FUNCTION_BLOCK FB_PointCorr
VAR PERSISTENT
  _fX_Pos, _fX_Ref : LREAL;   // x position (correction / reference)
  _fY_Pos, _fY_Ref : LREAL;   // y position (correction / reference)
END_VAR
VAR
  bCmd_X_minus : BOOL;    // command x minus
  bCmd_X_plus  : BOOL;    // command x plus
  bCmd_Y_minus : BOOL;    // command y minus
  bCmd_Y_plus  : BOOL;    // command y plus
  bAny         : BOOL;    // any pressed
  tSlow, tFast : TON;
  rTrig        : R_TRIG;
  nIncr        : LREAL;
  nBtnColor    : UDINT;
  // settings (init)
  _aName       : STRING(3);   // name of element
  _aUnit       : STRING(10);  // element intended [unit]
  _fX_Min, _fX_Max : LREAL;   // limit x
  _fY_Min, _fY_Max : LREAL;   // limit y
  _fIncrStep    : LREAL;      // incr. step slow (stay on button), fast *10
  _bButnInvertX, _bButnInvertY : BOOL;  // change buttons
  _bValInvertX, _bValInvertY   : BOOL;  // value *-1
END_VAR
VAR CONSTANT
  RED          : UDINT := 16#FFFF0000;
  GREEN        : UDINT := 16#FF00FF00;
END_VAR

bAny := bCmd_X_minus OR bCmd_X_plus OR bCmd_Y_minus OR bCmd_Y_plus;
rTrig(CLK:=bAny);
tSlow(IN:=bAny AND NOT tSlow.Q, PT:=T#500MS);
tFast(IN:=bAny AND NOT rTrig.Q, PT:=T#2S);

IF    tFast.Q AND tSlow.Q THEN nIncr := 10*_fIncrStep;
ELSIF tSlow.Q OR rTrig.Q THEN nIncr := _fIncrStep;
ELSE               nIncr := 0;
END_IF

nBtnColor := GREEN;
//    button pressed     increment +/-                show limit
IF    (bCmd_X_minus AND NOT _bButnInvertX) OR (bCmd_X_plus  AND _bButnInvertX) THEN _fX_Pos := _fX_Pos - nIncr; IF _fX_Pos<=_fX_Min THEN nBtnColor:=RED; END_IF
ELSIF (bCmd_X_plus  AND NOT _bButnInvertX) OR (bCmd_X_minus AND _bButnInvertX) THEN _fX_Pos := _fX_Pos + nIncr; IF _fX_Pos>=_fX_Max THEN nBtnColor:=RED; END_IF
ELSIF (bCmd_Y_minus AND NOT _bButnInvertY) OR (bCmd_Y_plus  AND _bButnInvertY) THEN _fY_Pos := _fY_Pos - nIncr; IF _fY_Pos<=_fY_Min THEN nBtnColor:=RED; END_IF
ELSIF (bCmd_Y_plus  AND NOT _bButnInvertY) OR (bCmd_Y_minus AND _bButnInvertY) THEN _fY_Pos := _fY_Pos + nIncr; IF _fY_Pos>=_fY_Max THEN nBtnColor:=RED; END_IF
END_IF

// apply limit
IF _fX_Pos<=_fX_Min THEN _fX_Pos:=_fX_Min; END_IF
IF _fX_Pos>=_fX_Max THEN _fX_Pos:=_fX_Max; END_IF
IF _fY_Pos<=_fY_Min THEN _fY_Pos:=_fY_Min; END_IF
IF _fY_Pos>=_fY_Max THEN _fY_Pos:=_fY_Max; END_IF

(*correction value in X*)
PROPERTY fX : LREAL
GET
fX := SEL(_bValInvertX, _fX_Pos, -1*_fX_Pos);
END_GET
END_PROPERTY

PROPERTY fX_Ref : LREAL
GET
fX_Ref := _fX_Ref;
END_GET
SET
_fX_Ref := fX_Ref;
END_SET
END_PROPERTY

(*correction value in Y*)
PROPERTY fY : LREAL
GET
fY := SEL(_bValInvertY, _fY_Pos, -1*_fY_Pos);
END_GET
END_PROPERTY

PROPERTY fY_Ref : LREAL
GET
fY_Ref := _fY_Ref;
END_GET
SET
_fY_Ref := fY_Ref;
END_SET
END_PROPERTY

METHOD init : BOOL
VAR_INPUT
  aName : STRING(3);       // name
  aUnit : STRING(10);      // display unit
  fX_Min, fX_Max : LREAL;  // Limits
  fY_Min, fY_Max : LREAL;  // Limits
  fIncrStep      : LREAL;  // Increment step (slow) VISU
  bButnInvertX, bButnInvertY : BOOL;  // change buttons
  bValInvertX,  bValInvertY  : BOOL;  // value *-1
END_VAR
_aName := aName;
_aUnit := aUnit;
_fX_Min := fX_Min; _fX_Max := fX_Max;
_fY_Min := fY_Min; _fY_Max := fY_Max;
_fIncrStep := fIncrStep;
_bButnInvertX := bButnInvertX;
_bButnInvertY := bButnInvertY;
_bValInvertX := bValInvertX;
_bValInvertY := bValInvertY;
END_METHOD

END_FUNCTION_BLOCK

(* stored: Version 1.1.0.1, ProductVersion 3.1.4024.3
   POU FB_PointCorr: Id {26dce410-3ea3-4f52-a45b-7e55ad528458}, SpecialFunc None
   Property fX: Id {525b6b57-3f78-4df9-8238-4b1829d37546}
   Get Get: Id {2dfc8c39-4fc0-4e95-a53d-3da45db26936}
   Property fX_Ref: Id {88a42ec6-eee5-4150-8b90-87a805146048}
   Get Get: Id {74654c86-ca8c-4a7a-8ea7-7f6f838d428e}
   Set Set: Id {ed71f6a4-2050-4ccf-82bf-2e474326bdfe}
   Property fY: Id {58fae2e8-1ba9-437b-8d17-701c295c3887}
   Get Get: Id {c1458e08-6817-492b-b919-4e53a7767d9d}
   Property fY_Ref: Id {7718ef6e-d7c5-4e02-9bb5-b5f9f83625f0}
   Get Get: Id {75beda1f-6937-4794-8088-2d2cc96f3309}
   Set Set: Id {ce0798df-87c4-4060-b253-b7b6b5e18fa6}
   Method init: Id {f9e13d1c-84a6-4c36-b358-d3b1f6d75c9a} *)
